TYPE ST_Axis :
STRUCT
	sAxis_Name		: STRING:='Axis Name';
	sAxis_Num		: INT;
	Status			: REFERENCE TO ST_AxisStatus;

	
	bPowerOn		: BOOL:=TRUE;
	bPowerOnN		: BOOL:=TRUE;
	bPowerOnP		: BOOL:=TRUE;
	bReset			: BOOL;
	bStop			: BOOL;
	bStopBusy		: BOOL;
	bError			: BOOL;
	
	bEnabled		: BOOL;

	bJogFw			: BOOL;
	bJogBw			: BOOL;
	fJogStep		: LREAL;
	fJogVelocity	: LREAL	:=10.000; //mm/sec	
	eJogMode		: E_JogMode:=E_JogMode.MC_JOGMODE_STANDARD_SLOW;
	eDirection		: MC_Direction:=MC_Direction.MC_Positive_Direction;



	
	fAccelaration	: LREAL :=1500.0; //mm/sec2
	fDeceleration	: LREAL :=1500.0; //mm/sec2
	fJerk			: LREAL :=2250.0; //mm/sec3
	fAggressionFactor: LREAL:=2000;

		
	fOverride		: LREAL :=100.0;
	
	fActPos			: LREAL;
	fActPosModulo	: LREAL;
	fActVelo		: LREAL;
	

	fReqPosAbs		: LREAL;
	fReqPosRel		: LREAL;
	fReqPosMod		: LREAL;
	fReqVelo		: LREAL; //common for move Velocity Absolute Relative and Modulo
	
	bMoveAbs		: BOOL;
	bMoveAbs2		: BOOL;
	bMoveRel		: BOOL;
	bMoveRel2		: BOOL;
	bMoveMod		: BOOL;
	bMoveMod2		: BOOL;
	bMoveVel		: BOOL;

	
	bMoveAbsDone	: BOOL;
	bMoveAbsDone2	: BOOL;
	bMoveRelDone	: BOOL;
	bMoveRelDone2	: BOOL;
	bMoveModDone	: BOOL;
	bMoveModDone2	: BOOL;
	bMoveVelDone	: BOOL;

	bMoveAbsBusy	: BOOL;
	bMoveAbsBusy2	: BOOL;
	bMoveRelBusy	: BOOL;
	bMoveRelBusy2	: BOOL;
	bMoveModBusy	: BOOL;
	bMoveModBusy2	: BOOL;
	bMoveVelBusy	: BOOL;
	
	bHome			: BOOL;
	bHomeSen		: BOOL; //sensor homming
	bHomeDone		: BOOL;
	bHomeBusy		: BOOL;
	bHomeMode_Direct: BOOL;
	eHomeMode		: MC_HomingMode;
	
	iErrorDI		: WORD; // From Driver by SDO

END_STRUCT
END_TYPE

(* stored: Version 1.1.0.1, ProductVersion 3.1.4024.12
   DUT ST_Axis: Id {d94e9ce8-0a89-460b-b829-77534dd11c81} *)
